INTERFACE I_ControlBox

METHOD Joystick
VAR_INPUT
	eMode 	: E_Mode;
	eStatus : E_Status;
END_VAR
VAR_OUTPUT
	fJoystickY : LREAL;
END_VAR
END_METHOD

METHOD Lamps 
VAR_INPUT
	eMode 	: E_Mode;
	eStatus : E_Status;
END_VAR
END_METHOD

METHOD ModeSelector 
VAR_INPUT
END_VAR
VAR_OUTPUT
	eMode : E_Mode;
END_VAR
END_METHOD

METHOD PushButtons
VAR_INPUT
	eMode 	: E_Mode;
	eStatus : E_Status;
END_VAR
VAR_OUTPUT
	bStart : BOOL;
	bStop : BOOL;
END_VAR
END_METHOD

END_INTERFACE

(* stored: Version 1.1.0.1, ProductVersion 3.1.4024.10
   Itf I_ControlBox: Id {5c741758-32b4-4a5c-b560-a63e85cb966e}
   Method Joystick: Id {19e2a514-84b4-4626-9e10-2ea6911d1f91}
   Method Lamps: Id {705895e4-a55f-468b-bff0-8eb1edb6385c}
   Method ModeSelector: Id {602723b8-14f8-4c4d-9a3a-6c04bf063cdf}
   Method PushButtons: Id {29a30b71-236c-4f52-a1fd-80494c25ecbb} *)
